(* IEC 61131-3 sources: RAG_PLC/data/result/test/063, 2 files *)

(* ---- wrapped.st ---- *)
(* =========================================================
   Generated by PLC-Eval Benchmark Wrapper
   ========================================================= *)

FUNCTION_BLOCK LLM_Wrapper_FB
VAR_INPUT
    CB : BYTE;
    E : BOOL;
    PIN : STRING[8];
END_VAR

VAR_OUTPUT
    TP : BOOL;
END_VAR

VAR
    POS : INT := 1;
END_VAR

TP := FALSE;
IF E THEN
    IF CB = BYTE_TO_INT(GET_CHAR(PIN, POS)) THEN
        POS := POS + 1;
        IF POS > LEN(PIN) THEN
            (* 检测到正确的代码 *)
            TP := TRUE;
            POS := 1;
        END_IF;
    ELSE
        POS := 1;
    END_IF;
END_IF;
END_FUNCTION_BLOCK

PROGRAM Auto_Proxy_Prg
  VAR
    instance : LLM_Wrapper_FB;
  END_VAR

  instance();
END_PROGRAM

CONFIGURATION Config0
  RESOURCE Res0 ON PLC
    TASK TaskMain(INTERVAL := T#20ms, PRIORITY := 0);
    PROGRAM Inst0 WITH TaskMain : Auto_Proxy_Prg;
  END_RESOURCE
END_CONFIGURATION

(* ---- raw_code.st ---- *)
VAR_INPUT
    CB : BYTE;
    E : BOOL;
    PIN : STRING[8];
END_VAR

VAR_OUTPUT
    TP : BOOL;
END_VAR

VAR
    POS : INT := 1;
END_VAR

TP := FALSE;
IF E THEN
    IF CB = BYTE_TO_INT(GET_CHAR(PIN, POS)) THEN
        POS := POS + 1;
        IF POS > LEN(PIN) THEN
            (* 检测到正确的代码 *)
            TP := TRUE;
            POS := 1;
        END_IF;
    ELSE
        POS := 1;
    END_IF;
END_IF;
